Universal Robots PolyScope program: tete de mat2.urp

Program tete de mat2 (installation=LVP3 tete de mat essai2 directory=/programs/Soudure 2023_03_27/V2.1 createdIn=5.9.4.1031232 lastSavedIn=5.11.9.1010452 robotSerialNumber=20225200921)
Calibrated DH parameters: a=[-0.00003, -0.368557, -0.560435, 0, -0.000026, 0]; d=[0.180818, -449.783649, 477.665205, -27.707784, 0.119652, 0.115612]; alpha=[1.571383, 0.001086, 0.003988, 1.568685, -1.571248, 0]; deltaTheta=[-0.000001, -0.924567, 7.403594, -0.195847, 0.000002, 0]
InitVariablesNode variables(variable(name=Test_Gaz, expression=False), variable(name=Test_Job, expression=False), variable(name=Test_Ordre_Mar, expression=False), variable(name=Valide_Gaz, expression=False), variable(name=fin_soud, expression=1), variable(name=secu_d, expression=0), variable(name=secu_g, expression=0), variable(name=timer_ret_gaz, expression=0))
BeforeStart
  Folder fonctions [hidden by the author, left out]
Robot Program (runOnlyOnce=false)
  SuppressedNode
    Folder Initialisation
      Loop Counting (count=1) loopVariable(name=Boucle_10)
        Script: fun_adresse_bp()
  SuppressedNode
    MoveJ speed 60 deg/s, acceleration 80 deg/s^2 (useActiveTCP=true) feature=Base
      SafeHome (positionOptionType=SPEED_AND_ACCELERATION speed=1.047198 acceleration=1.396263 nextMotionTime=2)
      Waypoint PointPassage (Variable): motionParameters(jointSpeed=0.523599 jointAcceleration=0.698132 cartesianSpeed=0.25 cartesianAcceleration=1.2); variable(featureName=Point_init_G)
      Waypoint PointPassage (Variable): motionParameters(jointSpeed=0.523599 jointAcceleration=0.698132 cartesianSpeed=0.25 cartesianAcceleration=1.2); variable(featureName=Point_Attente_G)
      Waypoint PointPassage (Variable): motionParameters(jointSpeed=0.523599 jointAcceleration=0.698132 cartesianSpeed=0.25 cartesianAcceleration=1.2); variable(featureName=Point_config_g)
      Waypoint PointPassage (Variable): motionParameters(jointSpeed=0.523599 jointAcceleration=0.698132 cartesianSpeed=0.25 cartesianAcceleration=1.2); variable(featureName=Point_Attente_G)
      Waypoint PointPassage (Variable): motionParameters(jointSpeed=0.523599 jointAcceleration=0.698132 cartesianSpeed=0.25 cartesianAcceleration=1.2); variable(featureName=Point_init_G)
      SafeHome (positionOptionType=SPEED_AND_ACCELERATION speed=1.047198 acceleration=1.396263 nextMotionTime=2)
      Waypoint PointPassage (Variable): motionParameters(jointSpeed=0.785398 jointAcceleration=1.047198 cartesianSpeed=0.25 cartesianAcceleration=1.2); variable(featureName=Point_avt_initD)
      Waypoint PointPassage (Variable): motionParameters(jointSpeed=0.523599 jointAcceleration=0.698132 cartesianSpeed=0.25 cartesianAcceleration=1.2); variable(featureName=Point_init_D)
      Waypoint PointPassage (Variable): motionParameters(jointSpeed=0.523599 jointAcceleration=0.698132 cartesianSpeed=0.25 cartesianAcceleration=1.2); variable(featureName=Point_Attente_D)
      Waypoint PointPassage (Variable): motionParameters(jointSpeed=0.523599 jointAcceleration=0.698132 cartesianSpeed=0.25 cartesianAcceleration=1.2); variable(featureName=Point_config_d)
      Waypoint PointPassage (Variable): motionParameters(jointSpeed=0.523599 jointAcceleration=0.698132 cartesianSpeed=0.25 cartesianAcceleration=1.2); variable(featureName=Point_Attente_D)
      Waypoint PointPassage (Variable): motionParameters(jointSpeed=0.523599 jointAcceleration=0.698132 cartesianSpeed=0.25 cartesianAcceleration=1.2); variable(featureName=Point_init_D)
      SafeHome (positionOptionType=SPEED_AND_ACCELERATION speed=1.047198 acceleration=1.396263 nextMotionTime=2)
  safe_mode := 0
  Folder Deplacement vers position initial
    SuppressedNode
      Popup Message (haltProgram=false message=debut deplacement vers position initiale inputType=Text)
    Set DigitalOutput pin=Cmd_Carter_Bit1; digitalValue=0
    Set DigitalOutput pin=Cmd_Carter_Bit2; digitalValue=0
    Loop While (checkContinuously=false) expression=SecuGaucheOk≟ True  or SecuDroiteOk≟ True
      Script: sync()
      'clingottement pour signifier qu'il y  un defaut sur un des carters '
      Set DigitalOutput pin=Dcy_Voyant; digitalValue=0
      Set DigitalOutput pin=Led_Arret; digitalValue=0
      Wait Sleep waitTime=0.5
      Set DigitalOutput pin=Dcy_Voyant; digitalValue=1
      Set DigitalOutput pin=Led_Arret; digitalValue=1
      Wait Sleep waitTime=0.5
    Set DigitalOutput pin=Led_Arret; digitalValue=0
    Set DigitalOutput pin=Dcy_Voyant; digitalValue=0
    Wait Sleep waitTime=2
    'etre sur de l'ouverture complete du carter '
    MoveL speed 0.2 mm/s, acceleration 10 mm/s^2 (useActiveTCP=true) feature=Base
      Waypoint PointPassage_12 (Relative): relativeFromPosition TCP in base x=100.468 y=319.613 z=576.47 mm, rx=-0.0214 ry=-0.0122 rz=1.5415 rad; joints [-139.419, 75.739, -163.156, -3.26, 89.083, -42.172] deg; TCP offset x=-8.331 y=2.512 z=301.573 mm, rx=0 ry=0 rz=0 rad; TCP in base x=100.463 y=319.639 z=576.462 mm, rx=-0.0214 ry=-0.0122 rz=1.5416 rad; joints [-139.419, 75.741, -163.155, -3.263, 89.08, -42.17] deg
      'Pos_cobot a etait affectuer a la position init (l3)'
      'Pos_cobot[2] correspond a la valeur Z de la postion init (l4)'
    SuppressedNode
      MoveJ speed 60 deg/s, acceleration 80 deg/s^2 (useActiveTCP=true) feature=Base
        SuppressedNode
          Waypoint Position_init: motionParameters(jointSpeed=1.047198 jointAcceleration=1.396263 cartesianSpeed=0.25 cartesianAcceleration=1.2); TCP in base x=96.613 y=317.698 z=575.432 mm, rx=-0.0254 ry=-0.0254 rz=1.5393 rad; joints [-139.566, 75.575, -163.284, -3.665, 88.92, -42.143] deg; TCP offset x=-6.782 y=1.742 z=298.685 mm, rx=0 ry=0 rz=0 rad
        SuppressedNode
          Waypoint PointPassage (Variable): variable(featureName=Point_init)
        'Apres avoir eu la position du robot et tester la valeur de Z pour faire un mouvement verticale on envoi le robot en position init'
    angle_base := get_actual_joint_positions()
    If angle_base[0] ≤0.7
      If angle_base[0]≥1.6
        SafeHome (positionOptionType=SPEED_AND_ACCELERATION speed=1.047198 acceleration=1.396263 nextMotionTime=2)
      ElseIf angle_base[0]>1.6
        MoveJ speed 100 deg/s, acceleration 80 deg/s^2 (useActiveTCP=true) feature=Base
          Waypoint PointPassage (Variable): variable(featureName=Point_init_D)
          Waypoint PointPassage (Variable): variable(featureName=Point_avt_initD)
      ElseIf angle_base[0]<0.7
        MoveJ speed 100 deg/s, acceleration 80 deg/s^2 (useActiveTCP=true) feature=Base
          Waypoint PointPassage (Variable): variable(featureName=Point_init_G)
    ElseIf angle_base[0]>1.6
      MoveJ speed 100 deg/s, acceleration 80 deg/s^2 (useActiveTCP=true) feature=Base
        Waypoint PointPassage (Variable): variable(featureName=Point_init_D)
        Waypoint PointPassage (Variable): variable(featureName=Point_avt_initD)
    ElseIf angle_base[0]<0.7
      MoveJ speed 100 deg/s, acceleration 80 deg/s^2 (useActiveTCP=true) feature=Base
        Waypoint PointPassage (Variable): variable(featureName=Point_init_G)
    SafeHome (positionOptionType=SPEED_AND_ACCELERATION speed=1.047198 acceleration=1.396263 nextMotionTime=2)
    angle_base := get_actual_joint_positions()
  'mode config'
  If Mode_manu ≟ False  and config_reglage ≟ False
    If (config_g ≟ 1)  and  (config_d ≟ 1)
      Script: pop_up_config_g_et_d()
    ElseIf (config_g ≟1)
      Script: pop_up_config_g()
    ElseIf config_d ≟ 1
      Script: pop_up_config_d()
    ElseIf (config_g ≟ 0) and (config_d ≟ 0)
      Script: pop_up_config()
    boucle := 1
    Loop While (checkContinuously=false) expression=(Mode_manu ≟ False ) and (boucle ≟ 1)  and (config_reglage≟ False )
      Loop While (checkContinuously=true) expression=Pret_Table_Droi≟ False  and Pret_Table_Gauc≟ False  and Mode_manu ≟  False  and config_reglage≟ False
        Set DigitalOutput pin=Voyant_Table_Ga; digitalValue=1
        Set DigitalOutput pin=Voyant_Table_Dr; digitalValue=0
        Wait Sleep waitTime=0.5
        Set DigitalOutput pin=Voyant_Table_Ga; digitalValue=0
        Set DigitalOutput pin=Voyant_Table_Dr; digitalValue=1
        Wait Sleep waitTime=0.5
        Script: sync()
      If Pret_Table_Gauc ≟ True
        Set DigitalOutput pin=Voyant_Table_Ga; digitalValue=1
        Set DigitalOutput pin=Voyant_Table_Dr; digitalValue=0
        'plus de demande du nombre de point a saisir'
        MoveJ speed 60 deg/s, acceleration 80 deg/s^2 (useActiveTCP=true) feature=Base
          Waypoint PointPassage (Variable): motionParameters(blendRadius=0.006); variable(featureName=Point_init_G)
          Waypoint PointPassage (Variable): motionParameters(blendRadius=0.006); variable(featureName=Point_Attente_G)
          Waypoint PointPassage (Variable): motionParameters(jointSpeed=0.523599 jointAcceleration=0.698132 cartesianSpeed=0.25 cartesianAcceleration=1.2); variable(featureName=Point_config_g)
          led_cobot := 1
          Script: fun_config_g()
          led_cobot := 0
          Script: fun_valid_config_g()
          MoveJ speed 60 deg/s, acceleration 80 deg/s^2 (useActiveTCP=true) feature=Base
            SuppressedNode
              Waypoint anti_poq_g: motionParameters(jointSpeed=0.523599 jointAcceleration=0.698132 cartesianSpeed=0.25 cartesianAcceleration=1.2 blendRadius=0.07); TCP in base x=433.126 y=153.22 z=577.202 mm, rx=0.0572 ry=-0.0147 rz=1.5652 rad; joints [-179.123, 70.738, -150.145, -9.057, 92.825, -1.059] deg; TCP offset x=-8.331 y=2.512 z=301.573 mm, rx=0 ry=0 rz=0 rad
            Waypoint PointPassage (Variable): motionParameters(blendRadius=0.006); variable(featureName=Point_Attente_G)
            Waypoint PointPassage (Variable): motionParameters(blendRadius=0.006); variable(featureName=Point_init_G)
            SuppressedNode
              Waypoint PointPassage (Variable): motionParameters(jointSpeed=0.523599 jointAcceleration=0.698132 cartesianSpeed=0.25 cartesianAcceleration=1.2); variable(featureName=Point_init)
            SafeHome (positionOptionType=SPEED_AND_ACCELERATION speed=1.047198 acceleration=1.396263 nextMotionTime=2)
      If Pret_Table_Droi ≟ True
        Set DigitalOutput pin=Voyant_Table_Dr; digitalValue=1
        Set DigitalOutput pin=Voyant_Table_Ga; digitalValue=0
        MoveJ speed 60 deg/s, acceleration 80 deg/s^2 (useActiveTCP=true) feature=Base
          Waypoint PointPassage (Variable): motionParameters(blendRadius=0.006); variable(featureName=Point_avt_initD)
          Waypoint PointPassage (Variable): variable(featureName=Point_init_D)
          Waypoint PointPassage (Variable): motionParameters(blendRadius=0.006); variable(featureName=Point_Attente_D)
          Waypoint PointPassage (Variable): motionParameters(jointSpeed=0.523599 jointAcceleration=0.698132 cartesianSpeed=0.25 cartesianAcceleration=1.2); variable(featureName=Point_config_d)
        led_cobot := 1
        Script: fun_config_d()
        led_cobot := 0
        Script: fun_valid_config_d()
        MoveJ speed 60 deg/s, acceleration 80 deg/s^2 (useActiveTCP=true) feature=Base
          SuppressedNode
            Waypoint anti_poq_1_d: motionParameters(jointSpeed=0.523599 jointAcceleration=0.698132 cartesianSpeed=0.25 cartesianAcceleration=1.2 blendRadius=0); TCP in base x=-432.081 y=47.828 z=581.386 mm, rx=0.0024 ry=-0.0004 rz=1.5709 rad; joints [-31.202, 71.743, -153.151, -8.683, 90.121, -148.72] deg
          SuppressedNode
            Waypoint anti_poq_2_d: motionParameters(jointSpeed=1.047198 jointAcceleration=1.396263 cartesianSpeed=0.25 cartesianAcceleration=1.2 blendRadius=0.07); TCP in base x=-292.604 y=310.313 z=583.956 mm, rx=-0.0324 ry=-0.0877 rz=3.0963 rad; joints [-72.124, 71.739, -151.869, -12.519, 87.987, -20.279] deg; TCP offset x=-8.331 y=2.512 z=301.573 mm, rx=0 ry=0 rz=0 rad
          SuppressedNode
            Waypoint PointPassage (Variable): motionParameters(jointSpeed=0.785398 jointAcceleration=1.047198 cartesianSpeed=0.25 cartesianAcceleration=1.2); variable(featureName=Point_init)
          Waypoint PointPassage (Variable): motionParameters(blendRadius=0.006); variable(featureName=Point_Attente_D)
          Waypoint PointPassage (Variable): motionParameters(blendRadius=0.006); variable(featureName=Point_init_D)
          Waypoint PointPassage (Variable): motionParameters(blendRadius=0.006); variable(featureName=Point_avt_initD)
          SafeHome (positionOptionType=SPEED_AND_ACCELERATION speed=1.047198 acceleration=1.396263 nextMotionTime=2)
  '"Reg"'
  If Mode_manu ≟ False  and config_reglage ≟ True
    If (config_g ≟ 1)  and  (config_d ≟ 1)
      Script: pop_up_reg_gd()
      boucle := 1
    ElseIf config_g ≟ 1
      Script: pop_up_reg_gd()
      boucle := 1
    ElseIf config_d ≟ 1
      Script: pop_up_reg_d()
      boucle := 1
    Else 
      Script: close_popup()
      Loop While (checkContinuously=false) expression=config_reglage ≟ True
        Popup Error (haltProgram=false message=Aucune configuration n'est actuellement detectée. inputType=Text)
    boucle := 1
    Loop While (checkContinuously=false) expression=(Mode_manu ≟ False ) and (boucle ≟ 1)  and (config_reglage≟ True )
      Loop While (checkContinuously=true) expression=Pret_Table_Droi≟ False  and Pret_Table_Gauc≟ False  and Mode_manu ≟  False  and config_reglage ≟ True
        If config_g ≟ 1
          Set DigitalOutput pin=Voyant_Table_Ga; digitalValue=1
        If config_d ≟ 1
          Set DigitalOutput pin=Voyant_Table_Dr; digitalValue=1
        Wait Sleep waitTime=0.5
        Set DigitalOutput pin=Voyant_Table_Ga; digitalValue=0
        Set DigitalOutput pin=Voyant_Table_Dr; digitalValue=0
        Wait Sleep waitTime=0.5
      If Pret_Table_Gauc ≟ True
        safe_mode := 1
        Set DigitalOutput pin=Voyant_Table_Ga; digitalValue=1
        Set DigitalOutput pin=Voyant_Table_Dr; digitalValue=0
        MoveJ speed 60 deg/s, acceleration 80 deg/s^2 (useActiveTCP=true) feature=Base
          Waypoint PointPassage (Variable): motionParameters(blendRadius=0.006); variable(featureName=Point_init_G)
          Waypoint PointPassage (Variable): motionParameters(blendRadius=0.006); variable(featureName=Point_Attente_G)
          Waypoint PointPassage (Variable): motionParameters(jointSpeed=0.523599 jointAcceleration=0.698132 cartesianSpeed=0.25 cartesianAcceleration=1.2); variable(featureName=pose_inter_g)
        led_cobot := 1
        Script: fun_Pas_A_Pas_g()
        led_cobot := 0
        safe_mode := 0
        boucle := 0
      If Pret_Table_Droi ≟ True
        safe_mode := 1
        Set DigitalOutput pin=Voyant_Table_Dr; digitalValue=1
        Set DigitalOutput pin=Voyant_Table_Ga; digitalValue=0
        MoveJ speed 60 deg/s, acceleration 80 deg/s^2 (useActiveTCP=true) feature=Base
          Waypoint PointPassage (Variable): motionParameters(blendRadius=0.006); variable(featureName=Point_avt_initD)
          Waypoint PointPassage (Variable): motionParameters(blendRadius=0.006); variable(featureName=Point_init_D)
          Waypoint PointPassage (Variable): motionParameters(jointSpeed=0.523599 jointAcceleration=0.698132 cartesianSpeed=0.25 cartesianAcceleration=1.2); variable(featureName=pose_inter_d)
        led_cobot := 1
        Script: fun_Pas_A_Pas_d()
        led_cobot := 0
        safe_mode := 0
        boucle := 0
  'mode exe'
  If Mode_manu ≟ True
    If (config_g ≟ 1)  and  (config_d ≟ 1)
      Script: pop_up_exe()
      boucle := 1
    ElseIf config_g ≟ 1
      Script: pop_up_exe_g()
      boucle := 1
    ElseIf config_d ≟ 1
      Script: pop_up_exe_d()
      boucle := 1
    Else 
      Script: close_popup()
      Loop While (checkContinuously=false) expression=Mode_manu ≟ True
        Popup Error (haltProgram=false message=Aucune programmation n'est actuellement detectée, veillez à programmer une pièce avant de vouloir l'éxécuter. inputType=Text)
    Loop While (checkContinuously=false) expression=( Mode_manu ≟ True )  and (boucle ≟ 1)
      Loop While (checkContinuously=true) expression=Pret_Table_Droi≟ False  and Pret_Table_Gauc≟ False  and Mode_manu≟ True
        If config_g ≟ 1
          Set DigitalOutput pin=Voyant_Table_Ga; digitalValue=1
        If config_d ≟ 1
          Set DigitalOutput pin=Voyant_Table_Dr; digitalValue=1
        Wait Sleep waitTime=0.5
        Set DigitalOutput pin=Voyant_Table_Ga; digitalValue=0
        Set DigitalOutput pin=Voyant_Table_Dr; digitalValue=0
        Wait Sleep waitTime=0.5
      If (Pret_Table_Gauc ≟ True ) and (config_g ≟ True )
        boucle_g := 1
        SuppressedNode
          Script: pop_up_deb_exe_g()
        Loop While (checkContinuously=false) expression=boucle_g ≟ 1
          Set DigitalOutput pin=Cmd_Carter_Bit1; digitalValue=1
          Set DigitalOutput pin=Voyant_Table_Ga; digitalValue=1
          Set DigitalOutput pin=Voyant_Table_Dr; digitalValue=0
          Wait Sleep waitTime=0.25
          Set DigitalOutput pin=Voyant_Table_Ga; digitalValue=0
          Wait Sleep waitTime=0.25
          If SecuGaucheOk ≟  False
            Set DigitalOutput pin=Voyant_Table_Ga; digitalValue=1
            SuppressedNode
              Wait Sleep waitTime=6
            If SecuGaucheOk ≟  False
              Script: close_popup()
              Wait DigitalInput pin=SecuGaucheOk; digitalValue=1
          If SecuGaucheOk ≟  True
            secu_g := 1
            Set DigitalOutput pin=Voyant_Table_Ga; digitalValue=1
            MoveJ speed 60 deg/s, acceleration 80 deg/s^2 (useActiveTCP=true) feature=Base
              Waypoint PointPassage (Variable): motionParameters(blendRadius=0.006); variable(featureName=Point_init_G)
              SuppressedNode
                Waypoint PointPassage (Variable): motionParameters(blendRadius=0.006); variable(featureName=Point_Attente_G)
            Script: fun_execution_g()
            MoveJ speed 60 deg/s, acceleration 80 deg/s^2 (useActiveTCP=true) feature=Base
              Waypoint PointPassage (Variable): motionParameters(blendRadius=0.006); variable(featureName=Point_Attente_G)
              Waypoint PointPassage (Variable): motionParameters(blendRadius=0.006); variable(featureName=Point_init_G)
              SafeHome (positionOptionType=SPEED_AND_ACCELERATION speed=1.047198 acceleration=1.396263 nextMotionTime=2)
            Set DigitalOutput pin=Cmd_Carter_Bit1; digitalValue=0
            secu_g := 0
            boucle_g := 0
        boucle := 0
      ElseIf (Pret_Table_Gauc ≟ True ) and (config_g ≟ False )
        Script: close_popup()
        Popup Error (haltProgram=false message=Aucune programmation n'est actuellement detectée sur la table gauche, veillez à programmer une pièce avant de vouloir l'éxécuter. inputType=Text)
        boucle := 0
      If (Pret_Table_Droi ≟ True ) and (config_d ≟ True )
        boucle_d := 1
        Script: pop_up_deb_exe_d()
        Loop While (checkContinuously=false) expression=boucle_d ≟ 1
          Set DigitalOutput pin=Cmd_Carter_Bit2; digitalValue=1
          Set DigitalOutput pin=Voyant_Table_Ga; digitalValue=0
          Set DigitalOutput pin=Voyant_Table_Dr; digitalValue=1
          Wait Sleep waitTime=0.25
          Set DigitalOutput pin=Voyant_Table_Dr; digitalValue=0
          Wait Sleep waitTime=0.25
          If SecuDroiteOk ≟  False
            Set DigitalOutput pin=Voyant_Table_Dr; digitalValue=1
            Wait Sleep waitTime=6
            If SecuDroiteOk ≟  False
              Script: close_popup()
              Wait DigitalInput pin=SecuDroiteOk; digitalValue=1
          If SecuDroiteOk ≟  True
            secu_d := 1
            Set DigitalOutput pin=Voyant_Table_Dr; digitalValue=1
            MoveJ speed 60 deg/s, acceleration 80 deg/s^2 (useActiveTCP=true) feature=Base
              Waypoint PointPassage (Variable): variable(featureName=Point_avt_initD)
              SuppressedNode
                Waypoint PointPassage (Variable): motionParameters(blendRadius=0.006); variable(featureName=Point_init_D)
            Script: fun_execution_d()
            Set DigitalOutput pin=Cmd_Carter_Bit2; digitalValue=0
            secu_d := 0
            boucle_d := 0
        boucle := 0
      ElseIf (Pret_Table_Droi ≟ True ) and (config_d ≟ False )
        Script: close_popup()
        Popup Error (haltProgram=false message=Aucune programmation n'est actuellement detectée sur la table droite, veillez à programmer une pièce avant de vouloir l'éxécuter. inputType=Text)
        boucle := 0
Thread Thread_1 (runOnlyOnce=false)
  Folder Test_Ordre_Marche [hidden by the author, left out]
  Script: sync()
Thread Thread_2 (runOnlyOnce=false)
  Folder mode_soudure [hidden by the author, left out]
  Script: sync()
Thread Thread_3 (runOnlyOnce=false)
  Folder led_cobot_2 [hidden by the author, left out]
  Script: sync()
Thread Thread_4 (runOnlyOnce=false)
  Folder led_cobot [hidden by the author, left out]
  Script: sync()
Thread Thread_5 (runOnlyOnce=false)
  Folder Test_Arc_On [hidden by the author, left out]
  Script: sync()
Thread Thread_6 (runOnlyOnce=false)
  Folder Test_Job
    If Test_Job≟ True
      SuppressedNode
        If Program_Soudure≟1 removedSiblings(If(type=ElseIf checkContinuously=false, expression=Program_Soudure≟2, children(Set(type=DigitalOutput, pin=Job_1, digitalValue=0), Set(type=DigitalOutput, pin=Job_2, digitalValue=1))), If(type=ElseIf checkContinuously=false, expression=Program_Soudure≟3, children(Set(type=DigitalOutput, pin=Job_1, digitalValue=1), Set(type=DigitalOutput, pin=Job_2, digitalValue=1))), If(type=ElseIf checkContinuously=false, expression=Program_Soudure≟4, children(Set(type=DigitalOutput, pin=Job_1, digitalValue=0), Set(type=DigitalOutput, pin=Job_2, digitalValue=0))), If(type=Else checkContinuously=false, children(Script(type=Line, expression=close_popup()), Popup(type=Error haltProgram=false message=Le Job soudure choisi n'existe pas. inputType=Text))))
          Set DigitalOutput pin=Job_1; digitalValue=1
          Set DigitalOutput pin=Job_2; digitalValue=0
      Test_Job := False
  Script: sync()
Thread Thread_7 (runOnlyOnce=false)
  Folder secu
    If SecuGaucheOk ≟  False  and secu_g ≟ 1
      Script: close_popup()
      Popup Error (haltProgram=true message=ATTENTION : Defaut carter ! inputType=Text)
    ElseIf SecuDroiteOk ≟ False  and secu_d ≟ 1
      Script: close_popup()
      Popup Error (haltProgram=true message=ATTENTION : Defaut carter ! inputType=Text)
  Script: sync()
Thread Thread_8 (runOnlyOnce=false)
  Folder bloq_soud_arret
    If Mode_soudure≟ False  and Test_Gaz ≟ True
      Script: close_popup()
      Popup Error (haltProgram=true message=Defaut : L'ordre de soudure a ete coupe pendant l'utilisation. inputType=Text)
  SuppressedNode
    Folder freedrive_droit
      If led_cobot ≟  True
        If tool_in[1] ≟ True
          Script: teach_mode()
        Else 
          Script: end_teach_mode()
  Script: sync()
SuppressedNode
  Thread Thread_9 (runOnlyOnce=false)
    Folder reglage
      If reglage_d ≠0
        Script file /programs/Programmes/cobot_v2/sript/Part_reglage/REGLAGE_D.script
          |     ##############################################################################
          | 
          | ########################soudure point#########################################
          | 
          |     ##############################################################################
          | 
          |         if reglage_d == 1:                                    #remplissage tableau
          |             teach_mode()
          |             fun_popup_soud(1, 1, i)
          |             fun_front_up(adresse_bp_cobot)
          |             tab_point_app_d[i] =  get_actual_tcp_pose()     #Enregistrer position dans tableau d'approche des soudue points quand appui bouton
          |             close_popup()
          | 
          |             fun_popup_soud(2, 1, i)
          |             fun_front_up(adresse_bp_cobot)
          |             tab_point_deb_d[i] =  get_actual_tcp_pose()     #Enregistrer position debut quand appui bouton bp_cobot
          |             close_popup()
          | 
          |             tab_point_ret_d[i] = tab_point_app_d[i]         #point de retrait est le meme que le point d approche
          |             end_teach_mode()
          |             global reconfig = 1
          |             global reglage_d = 0
          | 
          |             sync()
          | 
          |         ##############################################################################
          | 
          |     ##############################################################################
          | 
          | ########################soudure lineaire######################################
          | 
          |     ##############################################################################
          | 
          |         elif reglage_d == 2:                		            #remplissage tableau
          |             teach_mode()
          |             fun_popup_soud(1, 2, j)
          |             fun_front_up(adresse_bp_cobot)
          |             tab_lin_app_d[j] =  get_actual_tcp_pose()     	#Enregistrer position dans tableau d approche des soudures lineaire quand appui Bp_cobot
          |             close_popup()
          | 
          |             fun_popup_soud(2, 2, j)
          |             fun_front_up(adresse_bp_cobot)
          |             tab_lin_deb_d[j] =  get_actual_tcp_pose()     	#Enregistrer position dans tableau debut quand appui Bp_cobot
          |             close_popup()
          | 
          |             fun_popup_soud(6, 2, j)
          |             fun_front_up(adresse_bp_cobot)
          |             tab_lin_fin_d[j] =  get_actual_tcp_pose()     	#Enregistrer position dans un tableau fin quand appui Bp_cobot
          |             close_popup()
          | 
          |             vit_lin_d[j] = fun_demande_vit(2)
          | 
          |             fun_popup_soud(7, 2, j)
          |             fun_front_up(adresse_bp_cobot)
          |             tab_lin_ret_d[j] =  get_actual_tcp_pose()     	#Enregistrer position dans tableau retrait quand appui Bp_cobot
          |             close_popup()
          |             end_teach_mode()
          |             global reglage_d = 0
          | 
          |             sync()
          | 
          |         ##############################################################################
          | 
          |     ##############################################################################
          | 
          | #########################soudure arc de cercle##################################
          | 
          |     #################################################################################
          | 
          |         elif reglage_d == 3:                                  #remplissage tableau
          |             teach_mode()
          |             fun_popup_soud(1, 3, k)
          |             fun_front_up(adresse_bp_cobot)
          |             tab_arc_app_d[k] =  get_actual_tcp_pose() 	    #Enregistrer position dans tableau d approche des soudures arc de cercle quand appui
          |             close_popup()
          | 
          |             fun_popup_soud(2, 3, k)
          |             fun_front_up(adresse_bp_cobot)
          |             tab_arc_deb_d[k] =  get_actual_tcp_pose() 	    #Enregistrer position dans tableau debut quand appui Bp_d
          |             close_popup()
          | 
          |             fun_popup_soud(4, 3, k)
          |             fun_front_up(adresse_bp_cobot)
          |             tab_arc_mil_d[k] =  get_actual_tcp_pose() 	    #Enregistrer position dans tableau milieu quand appui Bp_cobot
          |             close_popup()
          | 
          |             fun_popup_soud(6, 3, k)
          |             fun_front_up(adresse_bp_cobot)
          |             tab_arc_fin_d[k] =  get_actual_tcp_pose() 	    #Enregistrer position dans un tableau fin quand appui Bp_cobot
          |             close_popup()
          | 
          |             vit_arc_d[k] = fun_demande_vit(3)               #demande de vitesse des soudures lineaire
          | 
          |             fun_popup_soud(7, 3, k)
          |             fun_front_up(adresse_bp_cobot)
          |             tab_arc_ret_d[k] =  get_actual_tcp_pose() 	    #Enregistrer position dans tableau retrait quand appui Bp_cobot
          |             close_popup()
          |             end_teach_mode()
          |             global reglage_d = 0
          | 
          |             sync()
          | 
          |         ##############################################################################
          | 
          |     ##############################################################################
          | 
          | ############################soudure cercle####################################
          | 
          |     #################################################################################
          | 
          |         elif reglage_d == 4:                                  #remplissage tableau
          |             teach_mode()
          |             fun_popup_soud(1, 4, l)
          |             fun_front_up(adresse_bp_cobot)
          |             tab_cer_app_d[l] =  get_actual_tcp_pose()     	#Enregistrer position dans tableau d approche des soudures arc de cercle quand appui Bp_cobot
          |             close_popup()
          | 
          |             fun_popup_soud(2, 4, l)
          |             fun_front_up(adresse_bp_cobot)
          |             tab_cer_deb_d[l] =  get_actual_tcp_pose()     	#Enregistrer position dans tableau debut quand appui Bp_cobot
          |             close_popup()
          | 
          |             fun_popup_soud(3, 4, l)
          |             fun_front_up(adresse_bp_cobot)
          |             tab_cer_quart_d[l] =  get_actual_tcp_pose()   	#Enregistrer position dans tableau d'approche des soudures arc de cercle quand appui Bp_d
          |             close_popup()
          | 
          |             fun_popup_soud(4, 4, l)
          |             fun_front_up(adresse_bp_cobot)
          |             tab_cer_mil_d[l] =  get_actual_tcp_pose()     	#Enregistrer position dans tableau milieu quand appui Bp_cobot
          |             close_popup()
          | 
          |             fun_popup_soud(5, 4, l)
          |             fun_front_up(adresse_bp_cobot)
          |             tab_cer_tro_d[l] =  get_actual_tcp_pose()     	#Enregistrer position dans tableau milieu quand appui Bp_cobot
          |             close_popup()
          | 
          |             fun_popup_soud(6, 4, l)
          |             fun_front_up(adresse_bp_cobot)
          |             tab_cer_fin_d[l] =  get_actual_tcp_pose()     	#Enregistrer position dans un tableau fin quand appui Bp_cobot
          |             close_popup()
          | 
          |             vit_cer_d[l] = fun_demande_vit(4)
          | 
          |             fun_popup_soud(7, 4, l)
          |             fun_front_up(adresse_bp_cobot)
          |             tab_cer_ret_d[l] =  get_actual_tcp_pose()    	#position de retrait est la meme que position d approche
          |             close_popup()
          |             end_teach_mode()
          |             global reglage_d = 0
          |             sync()
          | 
          |         end
          | 
          |     ##############################################################################
          | 
          | ############################################################
        Script: sync()
      If reglage_g ≠0
        Script file /programs/usbdisk_0/COBOT/finish/reg/REGLAGE_G.script
          |     ##############################################################################
          | 
          | ########################soudure point#########################################
          | 
          |     ##############################################################################
          | 
          |         if reglage_g == 1:                                    #remplissage tableau
          |             teach_mode()
          |             fun_popup_soud(1, 1, i)
          |             fun_front_up(adresse_bp_cobot)
          |             tab_point_app_g[i] =  get_actual_tcp_pose()     #Enregistrer position dans tableau d'approche des soudue points quand appui bouton
          |             close_popup()
          | 
          |             fun_popup_soud(2, 1, i)
          |             fun_front_up(adresse_bp_cobot)
          |             tab_point_deb_g[i] =  get_actual_tcp_pose()     #Enregistrer position debut quand appui bouton bp_cobot
          |             close_popup()
          | 
          |             tab_point_ret_g[i] = tab_point_app_g[i]         #point de retrait est le meme que le point d approche
          |             end_teach_mode()
          |             global reconfig = 1
          |             global reglage_g = 0
          | 
          |             sync()
          | 
          |         ##############################################################################
          | 
          |     ##############################################################################
          | 
          | ########################soudure lineaire######################################
          | 
          |     ##############################################################################
          | 
          |         elif reglage_g == 2:                		            #remplissage tableau
          |             teach_mode()
          |             fun_popup_soud(1, 2, j)
          |             fun_front_up(adresse_bp_cobot)
          |             tab_lin_app_g[j] =  get_actual_tcp_pose()     	#Enregistrer position dans tableau d approche des soudures lineaire quand appui Bp_cobot
          |             close_popup()
          | 
          |             fun_popup_soud(2, 2, j)
          |             fun_front_up(adresse_bp_cobot)
          |             tab_lin_deb_g[j] =  get_actual_tcp_pose()     	#Enregistrer position dans tableau debut quand appui Bp_cobot
          |             close_popup()
          | 
          |             fun_popup_soud(6, 2, j)
          |             fun_front_up(adresse_bp_cobot)
          |             tab_lin_fin_g[j] =  get_actual_tcp_pose()     	#Enregistrer position dans un tableau fin quand appui Bp_cobot
          |             close_popup()
          | 
          |             vit_lin_g[j] = fun_demande_vit(2)
          | 
          |             fun_popup_soud(7, 2, j)
          |             fun_front_up(adresse_bp_cobot)
          |             tab_lin_ret_g[j] =  get_actual_tcp_pose()     	#Enregistrer position dans tableau retrait quand appui Bp_cobot
          |             close_popup()
          |             end_teach_mode()
          |             global reglage_g = 0
          | 
          |             sync()
          | 
          |         ##############################################################################
          | 
          |     ##############################################################################
          | 
          | #########################soudure arc de cercle##################################
          | 
          |     #################################################################################
          | 
          |         elif reglage_g == 3:                                  #remplissage tableau
          |             teach_mode()
          |             fun_popup_soud(1, 3, k)
          |             fun_front_up(adresse_bp_cobot)
          |             tab_arc_app_g[k] =  get_actual_tcp_pose() 	    #Enregistrer position dans tableau d approche des soudures arc de cercle quand appui
          |             close_popup()
          | 
          |             fun_popup_soud(2, 3, k)
          |             fun_front_up(adresse_bp_cobot)
          |             tab_arc_deb_g[k] =  get_actual_tcp_pose() 	    #Enregistrer position dans tableau debut quand appui BP_cobot
          |             close_popup()
          | 
          |             fun_popup_soud(4, 3, k)
          |             fun_front_up(adresse_bp_cobot)
          |             tab_arc_mil_g[k] =  get_actual_tcp_pose() 	    #Enregistrer position dans tableau milieu quand appui Bp_cobot
          |             close_popup()
          | 
          |             fun_popup_soud(6, 3, k)
          |             fun_front_up(adresse_bp_cobot)
          |             tab_arc_fin_g[k] =  get_actual_tcp_pose() 	    #Enregistrer position dans un tableau fin quand appui Bp_cobot
          |             close_popup()
          | 
          |             vit_arc_g[k] = fun_demande_vit(3)               #demande de vitesse des soudures lineaire
          | 
          |             fun_popup_soud(7, 3, k)
          |             fun_front_up(adresse_bp_cobot)
          |             tab_arc_ret_g[k] =  get_actual_tcp_pose() 	    #Enregistrer position dans tableau retrait quand appui Bp_cobot
          |             close_popup()
          |             end_teach_mode()
          |             global reglage_g = 0
          | 
          |             sync()
          | 
          |         ##############################################################################
          | 
          |     ##############################################################################
          | 
          | ############################soudure cercle####################################
          | 
          |     #################################################################################
          | 
          |         elif reglage_g == 4:                                  #remplissage tableau
          |             teach_mode()
          |             fun_popup_soud(1, 4, l)
          |             fun_front_up(adresse_bp_cobot)
          |             tab_cer_app_g[l] =  get_actual_tcp_pose()     	#Enregistrer position dans tableau d approche des soudures arc de cercle quand appui Bp_cobot
          |             close_popup()
          | 
          |             fun_popup_soud(2, 4, l)
          |             fun_front_up(adresse_bp_cobot)
          |             tab_cer_deb_g[l] =  get_actual_tcp_pose()     	#Enregistrer position dans tableau debut quand appui Bp_cobot
          |             close_popup()
          | 
          |             fun_popup_soud(3, 4, l)
          |             fun_front_up(adresse_bp_cobot)
          |             tab_cer_quart_g[l] =  get_actual_tcp_pose()   	#Enregistrer position dans tableau d'approche des soudures arc de cercle quand appui Bp_cobot
          |             close_popup()
          | 
          |             fun_popup_soud(4, 4, l)
          |             fun_front_up(adresse_bp_cobot)
          |             tab_cer_mil_g[l] =  get_actual_tcp_pose()     	#Enregistrer position dans tableau milieu quand appui Bp_cobot
          |             close_popup()
          | 
          |             fun_popup_soud(5, 4, l)
          |             fun_front_up(adresse_bp_cobot)
          |             tab_cer_tro_g[l] =  get_actual_tcp_pose()     	#Enregistrer position dans tableau milieu quand appui Bp_cobot
          |             close_popup()
          | 
          |             fun_popup_soud(6, 4, l)
          |             fun_front_up(adresse_bp_cobot)
          |             tab_cer_fin_g[l] =  get_actual_tcp_pose()     	#Enregistrer position dans un tableau fin quand appui Bp_cobot
          |             close_popup()
          | 
          |             vit_cer_g[l] = fun_demande_vit(4)
          | 
          |             fun_popup_soud(7, 4, l)
          |             fun_front_up(adresse_bp_cobot)
          |             tab_cer_ret_g[l] =  get_actual_tcp_pose()    	#position de retrait est la meme que position d approche
          |             close_popup()
          |             end_teach_mode()
          |             global reglage_g = 0
          |             sync()
          | 
          |         end
          | 
          |     ##############################################################################
          | 
          | ############################################################
        Script: sync()
      Script: sync()
    Script: sync()
Thread Thread_10 (runOnlyOnce=false)
  Folder reglage [hidden by the author, left out]
  Script: sync()
